// TIA Portal V20 export
// export: Created 2025-12-01T14:57:25.6351868Z, ExportSetting None, DisplayName Totally Integrated Automation Portal, DisplayVersion V20 Update 3, DisplayName TIA Portal Openness, DisplayVersion V20 Update 3, DisplayName TIA Portal Version Control Interface, DisplayVersion V20 Update 3, DisplayName STEP 7 Professional, DisplayVersion V20 Update 3, DisplayName STEP 7 Safety, DisplayVersion V20 Update 2, DisplayName WinCC Basic/Comfort/Advanced, DisplayVersion V20 Update 3, DisplayName WinCC Professional, DisplayVersion V20 Update 3, DisplayName WinCC Unified, DisplayVersion V20 Update 3
FUNCTION_BLOCK "FB483_Interlock_IKPAL_Paletas"   // FB483, LAD
{ S7_Optimized_Access := 'FALSE' }
// stored: AutoNumber false, SetENOAutomatically false
   VAR_INPUT
      MesaPreformado : UInt;
      MesaVacios : UInt;
      MesaPaleta : UInt;
      Dir_Inicial : UInt;
      Nodo_OK : Bool;
      AvisoPreformado_PRV : Bool;
      OrdenMarchaPreformado_PRV : Bool;
      AvisoPreformado_PRV_Manual_AV : Bool;
      AvisoPreformado_PRV_Manual_Ret : Bool;
      PermisoExtenderHorquilla : Bool;
      PermisoCentrarHorquilla : Bool;
      MaquetaArriba : Bool;
      MaquetaAbajo : Bool;
      PermisoPaleta_NXT : Bool;
      FinPaleta_NXT : Bool;
      PermisoPaleta_NXT_Manual_Av : Bool;
      PermisoPaleta_NXT_Manual_Ret : Bool;
      PermisoÂperturaPuertas : Bool;
   END_VAR
   VAR_OUTPUT
      EstadoIKPAL : "EstadoZona";
      PermisoPreformado_PRV : Bool;
      FinPreformado_PRV : Bool;
      PermisoPreformado_PRV_Manual_AV : Bool;
      PermisoPreformado_PRV_Manual_Ret : Bool;
      PeticionPaletaVacia : Bool;
      HorquillasExtendidas : Bool;
      HorquillasCentradas : Bool;
      SubirMaqueta_Manual : Bool;
      BajarMaqueta_Manual : Bool;
      AvisoPaleta_NXT : Bool;
      OrdenMarchaPaleta_NXT : Bool;
      AvisoPaleta_NXT_Manual_AV : Bool;
      AvisoPaleta_NXT_Manual_Ret : Bool;
      PeticionAperturaPuertas : Bool;
      PuertasAccesoAbiertas : Bool;
   END_VAR
   VAR
      IKPAL_PLC { S7_SetPoint := 'True'} : "Interlock_Paletas_IKPAL_PLC";
      PLC_IKPAL { S7_SetPoint := 'True'} : "Interlock_Paletas_PLC_IKPAL";
      TIM_KeepAlive { S7_SetPoint := 'True'} : TON_TIME;
      Var_MesaPreformado : Struct
         ControlUT { S7_SetPoint := 'True'} : "UDT_UTs_Control";
         DatosUT { S7_SetPoint := 'True'} : "UDT_UTs_Datos";
         EtiquetaUT { S7_SetPoint := 'True'} : "UDT_UTs_Etiqueta";
      END_STRUCT;
      Var_MesaVacios : Struct
         ControlUT { S7_SetPoint := 'True'} : "UDT_UTs_Control";
         DatosUT { S7_SetPoint := 'True'} : "UDT_UTs_Datos";
         EtiquetaUT { S7_SetPoint := 'True'} : "UDT_UTs_Etiqueta";
      END_STRUCT;
      UT_MesaPreformado { ExternalAccessible := 'False'; ExternalVisible := 'False'; ExternalWritable := 'False'} : UInt;
      CotaAlturaPreformado : UInt;
      Matricula_Preformado : Array[1..10] of Byte;
      Mckey_Preformado : Array[1..8] of Byte;
      UT_MesaVacios { ExternalAccessible := 'False'; ExternalVisible := 'False'; ExternalWritable := 'False'} : UInt;
      Matricula_Vacios : Array[1..10] of Byte;
      Mckey_Vacios : Array[1..8] of Byte;
      Matricula_Paleta : Array[1..10] of Byte;
      Mckey_Paleta : Array[1..8] of Byte;
      NumMckey_Paleta : DInt;
      IdentificadorUT_Paleta : UDInt;
      MemoKeepAlive : Bool;
      ExisteUT_Preformado : Bool;
      ExisteUT_Vacios : Bool;
   END_VAR
   VAR_TEMP
      EstadoMesaPreformado : "EstadoZona";
      EstadoMesaVacios : "EstadoZona";
      EstadoMesaPaleta : "EstadoZona";
      EstadoVIMesaPreformado : "EstadosMesa";
      EstadoVIMesaVacios : "EstadosMesa";
      EstadoVIMesaPaleta : "EstadosMesa";
      Interlock_Entradas : "Interlock_Paletas_IKPAL_PLC";
      Interlock_Salidas : "Interlock_Paletas_PLC_IKPAL";
      Guardar_AR1 : DWord;
      Guardar_AR2 : DWord;
      P_Entradas : Any;
      P_Salidas : Any;
      P_L_Entradas : Any;
      P_L_Salidas : Any;
      P_DI_Entradas : Any;
      P_DI_Salidas : Any;
      P_AnyTemporal : Any;
      P_Temporal : DWord;
      DBInstancia : Word;
      NumeroUT : UInt;
      LongMatricula : UInt;
      LongMckey : UInt;
      LongEntradas : UInt;
      LongSalidas : UInt;
      DBOrigen : UInt;
      DBDestino : UInt;
      OffsetOrigen : UInt;
      OffsetDestino : UInt;
      P_Origen : DWord;
      P_Destino : DWord;
      Valor : UDInt;
      Indice : UInt;
      IndiceMatricula : UInt;
      ReturnValor : Int;
      Cero : Byte;
      ErrorMaquinaAsociada : Bool;
      FlancoKeepAlive : Bool;
   END_VAR
   VAR_TEMP   // added for the SCL form of the ladder/FBD networks
      _w1 : Bool;
      _w2 : Bool;
   END_VAR
BEGIN

REGION Network 1: INICIALIZAR
END_REGION

REGION Network 2: INICIALIZAR - Recoger las Variables de Estado de la Mesa de Preformado
   // Se recoge - Estado_CBx
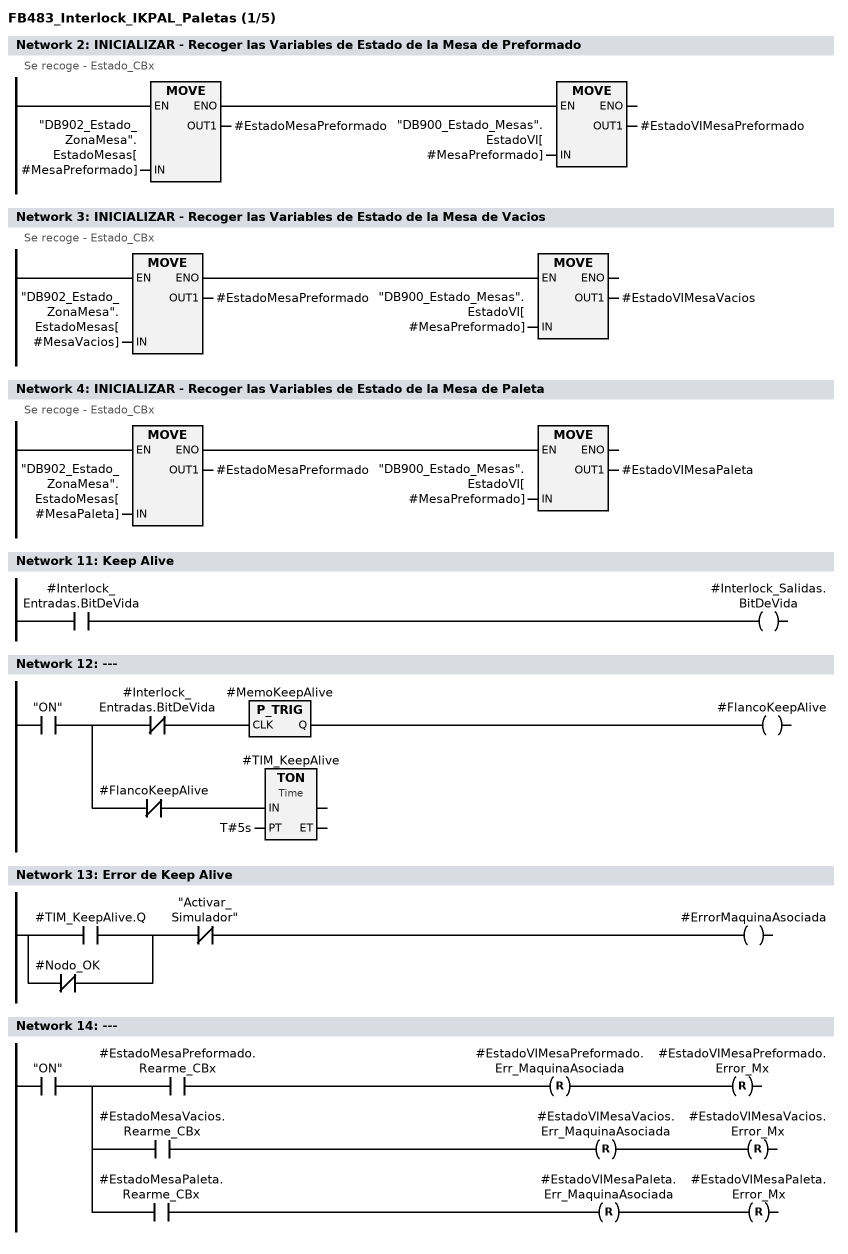
   RUNG wire#powerrail
      Move(in := "DB902_Estado_ZonaMesa".EstadoMesas[#MesaPreformado], out1 => #EstadoMesaPreformado)
      Move(in := "DB900_Estado_Mesas".EstadoVI[#MesaPreformado], out1 => #EstadoVIMesaPreformado)
   END_RUNG
   // the same network as SCL:
   #EstadoMesaPreformado := "DB902_Estado_ZonaMesa".EstadoMesas[#MesaPreformado];
   #EstadoVIMesaPreformado := "DB900_Estado_Mesas".EstadoVI[#MesaPreformado];
END_REGION

REGION Network 3: INICIALIZAR - Recoger las Variables de Estado de la Mesa de Vacios
   // Se recoge - Estado_CBx
   RUNG wire#powerrail
      Move(in := "DB902_Estado_ZonaMesa".EstadoMesas[#MesaVacios], out1 => #EstadoMesaPreformado)
      Move(in := "DB900_Estado_Mesas".EstadoVI[#MesaPreformado], out1 => #EstadoVIMesaVacios)
   END_RUNG
   // the same network as SCL:
   #EstadoMesaPreformado := "DB902_Estado_ZonaMesa".EstadoMesas[#MesaVacios];
   #EstadoVIMesaVacios := "DB900_Estado_Mesas".EstadoVI[#MesaPreformado];
END_REGION

REGION Network 4: INICIALIZAR - Recoger las Variables de Estado de la Mesa de Paleta
   // Se recoge - Estado_CBx
   RUNG wire#powerrail
      Move(in := "DB902_Estado_ZonaMesa".EstadoMesas[#MesaPaleta], out1 => #EstadoMesaPreformado)
      Move(in := "DB900_Estado_Mesas".EstadoVI[#MesaPreformado], out1 => #EstadoVIMesaPaleta)
   END_RUNG
   // the same network as SCL:
   #EstadoMesaPreformado := "DB902_Estado_ZonaMesa".EstadoMesas[#MesaPaleta];
   #EstadoVIMesaPaleta := "DB900_Estado_Mesas".EstadoVI[#MesaPreformado];
END_REGION

NETWORK
TITLE = Inicializar Variables Internas del Programa
//////////////////////////////////////////////////////////////////////////////
/// Inicializar las variables que necesita la FB

      L     56;  // Longitud de las Entradas
      T     #LongEntradas;
      L     56;  // Longitud de las Salidas
      T     #LongSalidas;
      L     10;  // Longitud de la Matricula
      T     #LongMatricula;
      L     8;  // Longitud del Mckey
      T     #LongMckey;

      L     DINO;  // Numero del DB de Instancia
      T     #DBInstancia;




NETWORK
TITLE = Preparacion de Punteros Any de las Entradas y Salidas
//////////////////////////////////////////////////////////////////////////////

      TAR1  #Guardar_AR1;  // Guardar AR1


//////////////////////////////////////////////////////////////////////////////
/// Puntero Any a las Entradas y Salidas (Temporales)

      LAR1  P##P_L_Entradas;  // - Any - Entradas del interlock
      L     B#16#10;  //   10H para S7
      T     LB [AR1, P#0.0];
      L     B#16#2;  //   Tipo de Datos (BYTE)
      T     LB [AR1, P#1.0];
      L     #LongEntradas;  //   Cantidad de datos
      T     LW [AR1, P#2.0];
      L     0;  //   Numero de DB (Temporal = 0)
      T     LW [AR1, P#4.0];
      L     P##Interlock_Entradas;  //   Direccion de Inicio
      T     LD [AR1, P#6.0];
      L     B#16#87;  //   El Area de Memoria = Temporal (Nota: No 86)
      T     LB [AR1, P#6.0];


      LAR1  P##P_L_Salidas;  // - Any - Salidas del interlock
      L     B#16#10;  //   10H para S7
      T     LB [AR1, P#0.0];
      L     B#16#2;  //   Tipo de Datos (BYTE)
      T     LB [AR1, P#1.0];
      L     #LongSalidas;  //   Cantidad de datos
      T     LW [AR1, P#2.0];
      L     0;  //   Numero de DB (Temporal = 0)
      T     LW [AR1, P#4.0];
      L     P##Interlock_Salidas;  //   Direccion de Inicio
      T     LD [AR1, P#6.0];
      L     B#16#87;  //   El Area de Memoria = Temporal (Nota: No 86)
      T     LB [AR1, P#6.0];


//////////////////////////////////////////////////////////////////////////////
/// Puntero Any a las Entradas y Salidas (DB de Instancia)

      LAR1  P##P_DI_Entradas;  // - Any - Entradas del interlock
      L     B#16#10;  //   10H para S7
      T     LB [AR1, P#0.0];
      L     B#16#2;  //   Tipo de Datos (BYTE)
      T     LB [AR1, P#1.0];
      L     #LongEntradas;  //   Cantidad de datos
      T     LW [AR1, P#2.0];
      L     #DBInstancia;  //   Numero de DB de Instancia
      T     LW [AR1, P#4.0];
      L     P##IKPAL_PLC;  //   Direccion de Inicio
      T     LD [AR1, P#6.0];
      L     B#16#84;  //   El Area de Memoria = DB Instancia
      T     LB [AR1, P#6.0];

      LAR1  P##P_DI_Salidas;  // - Any - Salidas del interlock
      L     B#16#10;  //   10H para S7
      T     LB [AR1, P#0.0];
      L     B#16#2;  //   Tipo de Datos (BYTE)
      T     LB [AR1, P#1.0];
      L     #LongSalidas;  //   Cantidad de datos
      T     LW [AR1, P#2.0];
      L     #DBInstancia;  //   Numero de DB de Instancia
      T     LW [AR1, P#4.0];
      L     P##PLC_IKPAL;  //   Direccion de Inicio
      T     LD [AR1, P#6.0];
      L     B#16#84;  //   El Area de Memoria = DB Instancia
      T     LB [AR1, P#6.0];


//////////////////////////////////////////////////////////////////////////////
/// Puntero Any - De Lectura y Escritura de QUBIQA

      LAR1  P##P_Entradas;  // - Any - Entradas del interlock
      L     B#16#10;  //   10H para S7
      T     LB [AR1, P#0.0];
      L     B#16#2;  //   Tipo de Datos (BYTE)
      T     LB [AR1, P#1.0];
      L     #LongEntradas;  //   Cantidad de datos
      T     LW [AR1, P#2.0];
      L     0;  //   Numero de DB (Temporal = 0)
      T     LW [AR1, P#4.0];
      L     #Dir_Inicial;  //   Direccion de Inicio
      SLD   3;
      T     LD [AR1, P#6.0];
      L     B#16#81;  //   El Area de Memoria = Entradas
      T     LB [AR1, P#6.0];

      LAR1  P##P_Salidas;  // - Any - Entradas del interlock
      L     B#16#10;  //   10H para S7
      T     LB [AR1, P#0.0];
      L     B#16#2;  //   Tipo de Datos (BYTE)
      T     LB [AR1, P#1.0];
      L     #LongSalidas;  //   Cantidad de datos
      T     LW [AR1, P#2.0];
      L     0;  //   Numero de DB (Temporal = 0)
      T     LW [AR1, P#4.0];
      L     #Dir_Inicial;  //   Direccion de Inicio
      SLD   3;
      T     LD [AR1, P#6.0];
      L     B#16#82;  //   El Area de Memoria = Salidas
      T     LB [AR1, P#6.0];

//////////////////////////////////////////////////////////////////////////////

      LAR1  #Guardar_AR1;  // Recuperar AR1



NETWORK
TITLE = Inicializacion de las Entradas y Salidas
//////////////////////////////////////////////////////////////////////////////
/// Inicializar el interlock (Variables Temporales)

      L     0;
      T     #Cero;

      CALL  FILL
      ( BVAL    := #Cero,
        RET_VAL := #ReturnValor,
        BLK     := #P_L_Entradas
      );  // Inicializo las Entradas

      CALL  FILL
      ( BVAL    := #Cero,
        RET_VAL := #ReturnValor,
        BLK     := #P_L_Salidas
      );  // Inicializo las Salidas



NETWORK
TITLE = Lectura de las Entradas
//////////////////////////////////////////////////////////////////////////////
/// Lectura de las Entradas

      SET;  // Comprobacion del Nodo
      AN    #Nodo_OK;
      AN    "Activar_Simulador";
      JC    NoLeerInterlock;

      CALL  UBLKMOV
      ( SRCBLK  := #P_Entradas,
        RET_VAL := #ReturnValor,
        DSTBLK  := #P_L_Entradas
      );


//////////////////////////////////////////////////////////////////////////////
/// Final Lectura de las Entradas

NoLeerInterlock:NOP   0;

      CALL  UBLKMOV
      ( SRCBLK  := #P_L_Entradas,
        RET_VAL := #ReturnValor,
        DSTBLK  := #P_DI_Entradas
      );  // Guardar el DB de Instancia



NETWORK
TITLE = Leer Datos de la UT de la Mesa de Preformado
//////////////////////////////////////////////////////////////////////////////
/// Incializacion inicial
      SET;  // De Inicio no existe UT
      R     #ExisteUT_Preformado;

      L     0;
      T     #UT_MesaPreformado;

      L     0;
      T     #Cero;
      CALL  FILL
      ( BVAL    := #Cero,
        RET_VAL := #ReturnValor,
        BLK     := #Var_MesaPreformado
      );

      SET;
      L     #MesaPreformado;  // Existe Mesa de Preformado ?
      L     0;
      ==I;
      JC    NoExiteUT_Preformado;


//////////////////////////////////////////////////////////////////////////////
/// Se mira si existe UT
      L     "DB810_ColasMesas".Colas[#MesaPreformado].UT_PrimeraMesa;
      T     #NumeroUT;
      L     0;
      ==I;
      JC    NoExiteUT_Preformado;

      SET;  // Existe UT en la Mesa
      S     #ExisteUT_Preformado;

      L     #NumeroUT;
      T     #UT_MesaPreformado;

      CALL  BLKMOV
      ( SRCBLK  := "DB812_UTs_Control".UT[#UT_MesaPreformado],
        RET_VAL := #ReturnValor,
        DSTBLK  := #Var_MesaPreformado.ControlUT
      );
      CALL  BLKMOV
      ( SRCBLK  := "DB815_UTs_Datos".UT[#UT_MesaPreformado],
        RET_VAL := #ReturnValor,
        DSTBLK  := #Var_MesaPreformado.DatosUT
      );
      CALL  BLKMOV
      ( SRCBLK  := "DB814_UTs_Etiqueta".UT[#MesaPreformado],
        RET_VAL := #ReturnValor,
        DSTBLK  := #Var_MesaPreformado.EtiquetaUT
      );


//////////////////////////////////////////////////////////////////////////////
/// Inicializo los datos de la UT que necesita el Interlock de IKPAL
      CALL  FILL
      ( BVAL    := #Cero,
        RET_VAL := #ReturnValor,
        BLK     := #Mckey_Preformado
      );  // Inicializo el Mckey

      CALL  FILL
      ( BVAL    := #Cero,
        RET_VAL := #ReturnValor,
        BLK     := #Matricula_Preformado
      );  // Inicializo la Matricula

//////////////////////////////////////////////////////////////////////////////
/// Copia el Cota Altura de la UT para el Interlock con IKPAL
      L     "DB815_UTs_Datos".UT[#UT_MesaPreformado].CotaAltura;
      T     #CotaAlturaPreformado;

//////////////////////////////////////////////////////////////////////////////
/// Copia el Mckey de la UT para el Interlock con IKPAL
      L     "DB812_UTs_Control".UT[#UT_MesaPreformado].Mckey;
      T     #Valor;

      L     #DBInstancia;
      T     #DBDestino;
      L     P##Mckey_Preformado;
      T     #P_Destino;
      SRD   3;
      L     #LongMckey;
      +I;
      L     1;
      -I;
      T     #OffsetDestino;

      CALL  "FC891_EtiqDInt_EtiqChar"
      ( DB_String   := #DBDestino,
        Long_String := #LongMckey,
        Offset_Ini  := #OffsetDestino,
        Valor       := #Valor
      );

      L     #LongMckey;
Copia_MckeyPreformado:T     #Indice;

      OPN   DB [#DBDestino];
      L     DBB [#P_Destino];
      L     '0';
      -I;
      OPN   DB [#DBDestino];
      T     DBB [#P_Destino];

      L     #P_Destino;
      L     P#1.0;
      +D;
      T     #P_Destino;

      L     #Indice;
      LOOP  Copia_MckeyPreformado;


//////////////////////////////////////////////////////////////////////////////
/// Copia la Matricula de la UT para el Interlock con IKPAL
      L     0;
      T     #IndiceMatricula;

      L     #DBInstancia;
      T     #DBDestino;
      L     P##Matricula_Preformado;
      T     #P_Destino;

      L     #LongMatricula;
Copia_MatriculaPreformado:T     #Indice;

      L     "DB814_UTs_Etiqueta".UT[#UT_MesaPreformado].Etiqueta[#IndiceMatricula];
      L     '0';
      -I;
      OPN   DB [#DBDestino];
      T     DBB [#P_Destino];

      L     #IndiceMatricula;
      L     1;
      +I;
      T     #IndiceMatricula;

      L     #P_Destino;
      L     P#1.0;
      +D;
      T     #P_Destino;

      L     #Indice;
      LOOP  Copia_MatriculaPreformado;


//////////////////////////////////////////////////////////////////////////////
NoExiteUT_Preformado:NOP   0;  // Final de la Lectura de Datos



NETWORK
TITLE = Leer Datos de la UT de la Mesa de Vacios
//////////////////////////////////////////////////////////////////////////////
/// Incializacion inicial
      SET;  // De Inicio no existe UT
      R     #ExisteUT_Vacios;

      L     0;
      T     #Cero;
      CALL  FILL
      ( BVAL    := #Cero,
        RET_VAL := #ReturnValor,
        BLK     := #Var_MesaVacios
      );


      SET;
      L     #MesaVacios;  // Existe Mesa de Preformado ?
      L     0;
      ==I;
      JC    NoExiteUT_Vacios;


//////////////////////////////////////////////////////////////////////////////
/// Se mira si existe UT
      L     "DB810_ColasMesas".Colas[#MesaVacios].UT_PrimeraMesa;
      T     #NumeroUT;
      L     0;
      ==I;
      JC    NoExiteUT_Vacios;

      SET;  // Existe UT en la Mesa
      S     #ExisteUT_Vacios;

      L     #NumeroUT;
      T     #UT_MesaVacios;

      CALL  BLKMOV
      ( SRCBLK  := "DB812_UTs_Control".UT[#UT_MesaVacios],
        RET_VAL := #ReturnValor,
        DSTBLK  := #Var_MesaVacios.ControlUT
      );
      CALL  BLKMOV
      ( SRCBLK  := "DB815_UTs_Datos".UT[#UT_MesaVacios],
        RET_VAL := #ReturnValor,
        DSTBLK  := #Var_MesaVacios.DatosUT
      );
      CALL  BLKMOV
      ( SRCBLK  := "DB814_UTs_Etiqueta".UT[#MesaVacios],
        RET_VAL := #ReturnValor,
        DSTBLK  := #Var_MesaVacios.EtiquetaUT
      );


//////////////////////////////////////////////////////////////////////////////
/// Inicializo los datos de la UT que necesita el Interlock de IKPAL
      CALL  FILL
      ( BVAL    := #Cero,
        RET_VAL := #ReturnValor,
        BLK     := #Mckey_Vacios
      );  // Inicializo el Mckey

      CALL  FILL
      ( BVAL    := #Cero,
        RET_VAL := #ReturnValor,
        BLK     := #Matricula_Vacios
      );  // Inicializo la Matricula


//////////////////////////////////////////////////////////////////////////////
/// Copia el Mckey de la UT para el Interlock con IKPAL
      L     "DB812_UTs_Control".UT[#UT_MesaVacios].Mckey;
      T     #Valor;

      L     #DBInstancia;
      T     #DBDestino;
      L     P##Mckey_Vacios;
      T     #P_Destino;
      SRD   3;
      L     #LongMckey;
      +I;
      L     1;
      -I;
      T     #OffsetDestino;

      CALL  "FC891_EtiqDInt_EtiqChar"
      ( DB_String   := #DBDestino,
        Long_String := #LongMckey,
        Offset_Ini  := #OffsetDestino,
        Valor       := #Valor
      );

      L     #LongMckey;
Copia_MckeyVacios:T     #Indice;

      OPN   DB [#DBDestino];
      L     DBB [#P_Destino];
      L     '0';
      -I;
      OPN   DB [#DBDestino];
      T     DBB [#P_Destino];

      L     #P_Destino;
      L     P#1.0;
      +D;
      T     #P_Destino;

      L     #Indice;
      LOOP  Copia_MckeyVacios;


//////////////////////////////////////////////////////////////////////////////
/// Copia la Matricula de la UT para el Interlock con IKPA
      L     0;
      T     #IndiceMatricula;

      L     #DBInstancia;
      T     #DBDestino;
      L     P##Matricula_Vacios;
      T     #P_Destino;

      L     #LongMatricula;
Copia_MatriculaVacios:T     #Indice;

      L     "DB814_UTs_Etiqueta".UT[#UT_MesaVacios].Etiqueta[#IndiceMatricula];
      L     '0';
      -I;
      OPN   DB [#DBDestino];
      T     DBB [#P_Destino];

      L     #IndiceMatricula;
      L     1;
      +I;
      T     #IndiceMatricula;

      L     #P_Destino;
      L     P#1.0;
      +D;
      T     #P_Destino;

      L     #Indice;
      LOOP  Copia_MatriculaVacios;


//////////////////////////////////////////////////////////////////////////////
NoExiteUT_Vacios:NOP   0;  // Final de la Lectura de Datos



REGION Network 11: Keep Alive
   RUNG wire#powerrail
      Contact( #Interlock_Entradas.BitDeVida )
      Coil( #Interlock_Salidas.BitDeVida )
   END_RUNG
   // the same network as SCL:
   #Interlock_Salidas.BitDeVida := #Interlock_Entradas.BitDeVida;
END_REGION

REGION Network 12: ---
   RUNG wire#powerrail
      Contact( "ON" )
      wire#w1
      I_Contact( #Interlock_Entradas.BitDeVida )
      P_Trig( #MemoKeepAlive )
      Coil( #FlancoKeepAlive )
   END_RUNG
   RUNG wire#w1
      I_Contact( #FlancoKeepAlive )
      { S7_Templates := "time_type := Time" } #TIM_KeepAlive.TON(pt := T#5s, et =>)
   END_RUNG
   // the same network as SCL:
   #_w1 := "ON" AND NOT #Interlock_Entradas.BitDeVida;
   #_w2 := #_w1 AND NOT #MemoKeepAlive;   // rising edge
   #MemoKeepAlive := #_w1;
   #FlancoKeepAlive := #_w2;
   #TIM_KeepAlive(IN := "ON" AND NOT #FlancoKeepAlive, PT := T#5s);   // TON
END_REGION

REGION Network 13: Error de Keep Alive
   RUNG wire#powerrail
      Contact( #TIM_KeepAlive.Q )
      wire#w1
      I_Contact( "Activar_Simulador" )
      Coil( #ErrorMaquinaAsociada )
   END_RUNG
   RUNG wire#powerrail
      I_Contact( #Nodo_OK )
   END_RUNG wire#w1
   // the same network as SCL:
   #ErrorMaquinaAsociada := (#TIM_KeepAlive.Q OR NOT #Nodo_OK) AND NOT "Activar_Simulador";
END_REGION

REGION Network 14: ---
   RUNG wire#powerrail
      Contact( "ON" )
      wire#w1
      Contact( #EstadoMesaPreformado.Rearme_CBx )
      R_Coil( #EstadoVIMesaPreformado.Err_MaquinaAsociada )
      R_Coil( #EstadoVIMesaPreformado.Error_Mx )
   END_RUNG
   RUNG wire#w1
      Contact( #EstadoMesaVacios.Rearme_CBx )
      R_Coil( #EstadoVIMesaVacios.Err_MaquinaAsociada )
      R_Coil( #EstadoVIMesaVacios.Error_Mx )
   END_RUNG
   RUNG wire#w1
      Contact( #EstadoMesaPaleta.Rearme_CBx )
      R_Coil( #EstadoVIMesaPaleta.Err_MaquinaAsociada )
      R_Coil( #EstadoVIMesaPaleta.Error_Mx )
   END_RUNG
   // the same network as SCL:
   IF "ON" AND #EstadoMesaPreformado.Rearme_CBx THEN
       #EstadoVIMesaPreformado.Err_MaquinaAsociada := FALSE;
       #EstadoVIMesaPreformado.Error_Mx := FALSE;
   END_IF;
   IF "ON" AND #EstadoMesaVacios.Rearme_CBx THEN
       #EstadoVIMesaVacios.Err_MaquinaAsociada := FALSE;
       #EstadoVIMesaVacios.Error_Mx := FALSE;
   END_IF;
   IF "ON" AND #EstadoMesaPaleta.Rearme_CBx THEN
       #EstadoVIMesaPaleta.Err_MaquinaAsociada := FALSE;
       #EstadoVIMesaPaleta.Error_Mx := FALSE;
   END_IF;
END_REGION

REGION Network 15: ---
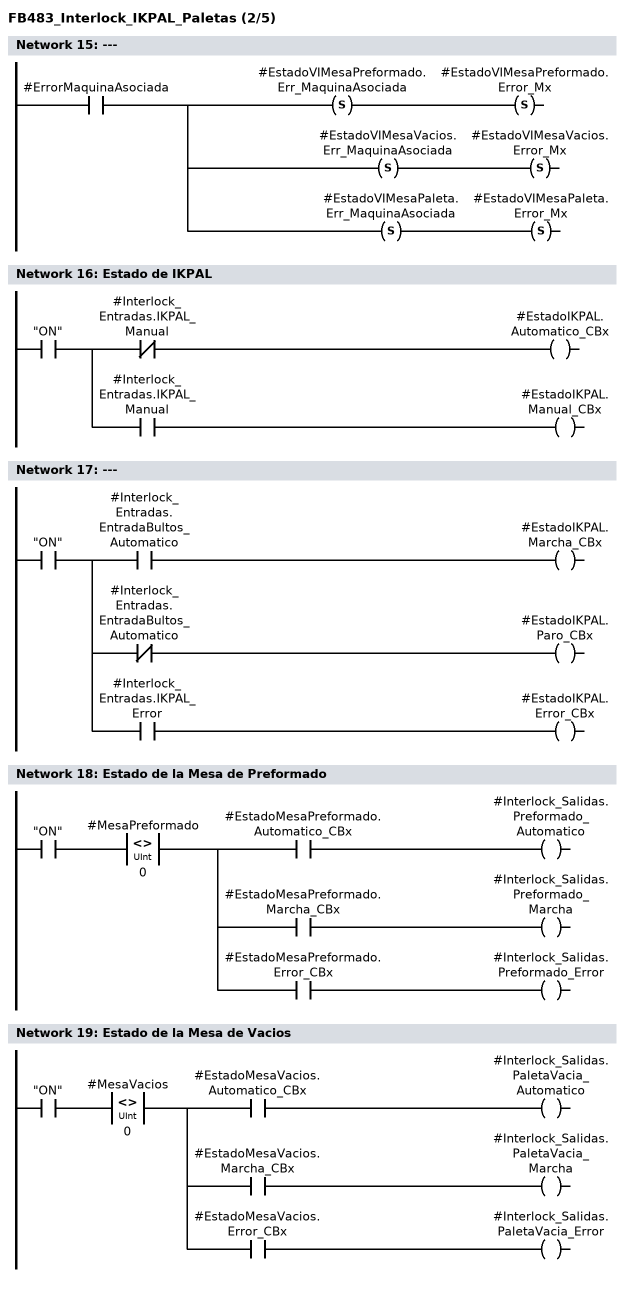
   RUNG wire#powerrail
      Contact( #ErrorMaquinaAsociada )
      wire#w1
      S_Coil( #EstadoVIMesaPreformado.Err_MaquinaAsociada )
      S_Coil( #EstadoVIMesaPreformado.Error_Mx )
   END_RUNG
   RUNG wire#w1
      S_Coil( #EstadoVIMesaVacios.Err_MaquinaAsociada )
      S_Coil( #EstadoVIMesaVacios.Error_Mx )
   END_RUNG
   RUNG wire#w1
      S_Coil( #EstadoVIMesaPaleta.Err_MaquinaAsociada )
      S_Coil( #EstadoVIMesaPaleta.Error_Mx )
   END_RUNG
   // the same network as SCL:
   IF #ErrorMaquinaAsociada THEN
       #EstadoVIMesaPreformado.Err_MaquinaAsociada := TRUE;
       #EstadoVIMesaPreformado.Error_Mx := TRUE;
       #EstadoVIMesaVacios.Err_MaquinaAsociada := TRUE;
       #EstadoVIMesaVacios.Error_Mx := TRUE;
       #EstadoVIMesaPaleta.Err_MaquinaAsociada := TRUE;
       #EstadoVIMesaPaleta.Error_Mx := TRUE;
   END_IF;
END_REGION

REGION Network 16: Estado de IKPAL
   RUNG wire#powerrail
      Contact( "ON" )
      wire#w1
      I_Contact( #Interlock_Entradas.IKPAL_Manual )
      Coil( #EstadoIKPAL.Automatico_CBx )
   END_RUNG
   RUNG wire#w1
      Contact( #Interlock_Entradas.IKPAL_Manual )
      Coil( #EstadoIKPAL.Manual_CBx )
   END_RUNG
   // the same network as SCL:
   #EstadoIKPAL.Automatico_CBx := "ON" AND NOT #Interlock_Entradas.IKPAL_Manual;
   #EstadoIKPAL.Manual_CBx := "ON" AND #Interlock_Entradas.IKPAL_Manual;
END_REGION

REGION Network 17: ---
   RUNG wire#powerrail
      Contact( "ON" )
      wire#w1
      Contact( #Interlock_Entradas.EntradaBultos_Automatico )
      Coil( #EstadoIKPAL.Marcha_CBx )
   END_RUNG
   RUNG wire#w1
      I_Contact( #Interlock_Entradas.EntradaBultos_Automatico )
      Coil( #EstadoIKPAL.Paro_CBx )
   END_RUNG
   RUNG wire#w1
      Contact( #Interlock_Entradas.IKPAL_Error )
      Coil( #EstadoIKPAL.Error_CBx )
   END_RUNG
   // the same network as SCL:
   #EstadoIKPAL.Marcha_CBx := "ON" AND #Interlock_Entradas.EntradaBultos_Automatico;
   #EstadoIKPAL.Paro_CBx := "ON" AND NOT #Interlock_Entradas.EntradaBultos_Automatico;
   #EstadoIKPAL.Error_CBx := "ON" AND #Interlock_Entradas.IKPAL_Error;
END_REGION

REGION Network 18: Estado de la Mesa de Preformado
   RUNG wire#powerrail
      Contact( "ON" )
      { S7_Templates := "SrcType := UInt" } NE_Contact(in1 := #MesaPreformado, in2 := 0)
      wire#w1
      Contact( #EstadoMesaPreformado.Automatico_CBx )
      Coil( #Interlock_Salidas.Preformado_Automatico )
   END_RUNG
   RUNG wire#w1
      Contact( #EstadoMesaPreformado.Marcha_CBx )
      Coil( #Interlock_Salidas.Preformado_Marcha )
   END_RUNG
   RUNG wire#w1
      Contact( #EstadoMesaPreformado.Error_CBx )
      Coil( #Interlock_Salidas.Preformado_Error )
   END_RUNG
   // the same network as SCL:
   #_w1 := "ON" AND (#MesaPreformado <> 0);
   #Interlock_Salidas.Preformado_Automatico := #_w1 AND #EstadoMesaPreformado.Automatico_CBx;
   #Interlock_Salidas.Preformado_Marcha := #_w1 AND #EstadoMesaPreformado.Marcha_CBx;
   #Interlock_Salidas.Preformado_Error := #_w1 AND #EstadoMesaPreformado.Error_CBx;
END_REGION

REGION Network 19: Estado de la Mesa de Vacios
   RUNG wire#powerrail
      Contact( "ON" )
      { S7_Templates := "SrcType := UInt" } NE_Contact(in1 := #MesaVacios, in2 := 0)
      wire#w1
      Contact( #EstadoMesaVacios.Automatico_CBx )
      Coil( #Interlock_Salidas.PaletaVacia_Automatico )
   END_RUNG
   RUNG wire#w1
      Contact( #EstadoMesaVacios.Marcha_CBx )
      Coil( #Interlock_Salidas.PaletaVacia_Marcha )
   END_RUNG
   RUNG wire#w1
      Contact( #EstadoMesaVacios.Error_CBx )
      Coil( #Interlock_Salidas.PaletaVacia_Error )
   END_RUNG
   // the same network as SCL:
   #_w1 := "ON" AND (#MesaVacios <> 0);
   #Interlock_Salidas.PaletaVacia_Automatico := #_w1 AND #EstadoMesaVacios.Automatico_CBx;
   #Interlock_Salidas.PaletaVacia_Marcha := #_w1 AND #EstadoMesaVacios.Marcha_CBx;
   #Interlock_Salidas.PaletaVacia_Error := #_w1 AND #EstadoMesaVacios.Error_CBx;
END_REGION

REGION Network 20: Estado de la Mesa de la Paleta
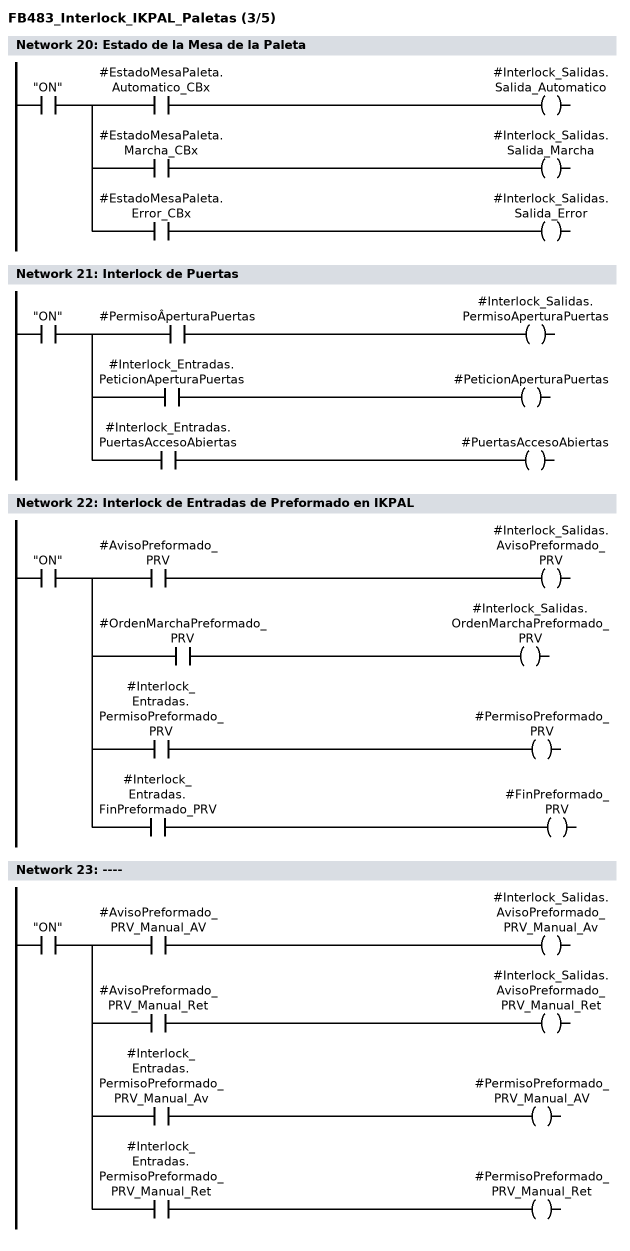
   RUNG wire#powerrail
      Contact( "ON" )
      wire#w1
      Contact( #EstadoMesaPaleta.Automatico_CBx )
      Coil( #Interlock_Salidas.Salida_Automatico )
   END_RUNG
   RUNG wire#w1
      Contact( #EstadoMesaPaleta.Marcha_CBx )
      Coil( #Interlock_Salidas.Salida_Marcha )
   END_RUNG
   RUNG wire#w1
      Contact( #EstadoMesaPaleta.Error_CBx )
      Coil( #Interlock_Salidas.Salida_Error )
   END_RUNG
   // the same network as SCL:
   #Interlock_Salidas.Salida_Automatico := "ON" AND #EstadoMesaPaleta.Automatico_CBx;
   #Interlock_Salidas.Salida_Marcha := "ON" AND #EstadoMesaPaleta.Marcha_CBx;
   #Interlock_Salidas.Salida_Error := "ON" AND #EstadoMesaPaleta.Error_CBx;
END_REGION

REGION Network 21: Interlock de Puertas
   RUNG wire#powerrail
      Contact( "ON" )
      wire#w1
      Contact( #PermisoÂperturaPuertas )
      Coil( #Interlock_Salidas.PermisoAperturaPuertas )
   END_RUNG
   RUNG wire#w1
      Contact( #Interlock_Entradas.PeticionAperturaPuertas )
      Coil( #PeticionAperturaPuertas )
   END_RUNG
   RUNG wire#w1
      Contact( #Interlock_Entradas.PuertasAccesoAbiertas )
      Coil( #PuertasAccesoAbiertas )
   END_RUNG
   // the same network as SCL:
   #Interlock_Salidas.PermisoAperturaPuertas := "ON" AND #PermisoÂperturaPuertas;
   #PeticionAperturaPuertas := "ON" AND #Interlock_Entradas.PeticionAperturaPuertas;
   #PuertasAccesoAbiertas := "ON" AND #Interlock_Entradas.PuertasAccesoAbiertas;
END_REGION

REGION Network 22: Interlock de Entradas de Preformado en IKPAL
   RUNG wire#powerrail
      Contact( "ON" )
      wire#w1
      Contact( #AvisoPreformado_PRV )
      Coil( #Interlock_Salidas.AvisoPreformado_PRV )
   END_RUNG
   RUNG wire#w1
      Contact( #OrdenMarchaPreformado_PRV )
      Coil( #Interlock_Salidas.OrdenMarchaPreformado_PRV )
   END_RUNG
   RUNG wire#w1
      Contact( #Interlock_Entradas.PermisoPreformado_PRV )
      Coil( #PermisoPreformado_PRV )
   END_RUNG
   RUNG wire#w1
      Contact( #Interlock_Entradas.FinPreformado_PRV )
      Coil( #FinPreformado_PRV )
   END_RUNG
   // the same network as SCL:
   #Interlock_Salidas.AvisoPreformado_PRV := "ON" AND #AvisoPreformado_PRV;
   #Interlock_Salidas.OrdenMarchaPreformado_PRV := "ON" AND #OrdenMarchaPreformado_PRV;
   #PermisoPreformado_PRV := "ON" AND #Interlock_Entradas.PermisoPreformado_PRV;
   #FinPreformado_PRV := "ON" AND #Interlock_Entradas.FinPreformado_PRV;
END_REGION

REGION Network 23: ----
   RUNG wire#powerrail
      Contact( "ON" )
      wire#w1
      Contact( #AvisoPreformado_PRV_Manual_AV )
      Coil( #Interlock_Salidas.AvisoPreformado_PRV_Manual_Av )
   END_RUNG
   RUNG wire#w1
      Contact( #AvisoPreformado_PRV_Manual_Ret )
      Coil( #Interlock_Salidas.AvisoPreformado_PRV_Manual_Ret )
   END_RUNG
   RUNG wire#w1
      Contact( #Interlock_Entradas.PermisoPreformado_PRV_Manual_Av )
      Coil( #PermisoPreformado_PRV_Manual_AV )
   END_RUNG
   RUNG wire#w1
      Contact( #Interlock_Entradas.PermisoPreformado_PRV_Manual_Ret )
      Coil( #PermisoPreformado_PRV_Manual_Ret )
   END_RUNG
   // the same network as SCL:
   #Interlock_Salidas.AvisoPreformado_PRV_Manual_Av := "ON" AND #AvisoPreformado_PRV_Manual_AV;
   #Interlock_Salidas.AvisoPreformado_PRV_Manual_Ret := "ON" AND #AvisoPreformado_PRV_Manual_Ret;
   #PermisoPreformado_PRV_Manual_AV := "ON" AND #Interlock_Entradas.PermisoPreformado_PRV_Manual_Av;
   #PermisoPreformado_PRV_Manual_Ret := "ON" AND #Interlock_Entradas.PermisoPreformado_PRV_Manual_Ret;
END_REGION

NETWORK
TITLE = ----
//////////////////////////////////////////////////////////////////
/// Copia de los datos de la Mesa de Preformado para IKPAL

      AN    #ExisteUT_Preformado;
      JC    FinalCopiaDatos_Preformado_IKPAL;

      L     #CotaAlturaPreformado;
      T     #Interlock_Salidas.CotaAlturaPreformado;

      CALL  UBLKMOV
      ( SRCBLK  := #Mckey_Preformado,
        RET_VAL := #ReturnValor,
        DSTBLK  := #Interlock_Salidas.MckeyPreformado
      );
      CALL  UBLKMOV
      ( SRCBLK  := #Matricula_Preformado,
        RET_VAL := #ReturnValor,
        DSTBLK  := #Interlock_Salidas.MatriculaPreformado
      );

FinalCopiaDatos_Preformado_IKPAL:NOP   0;



REGION Network 25: Interlock de Entradas de Vacios en IKPAL
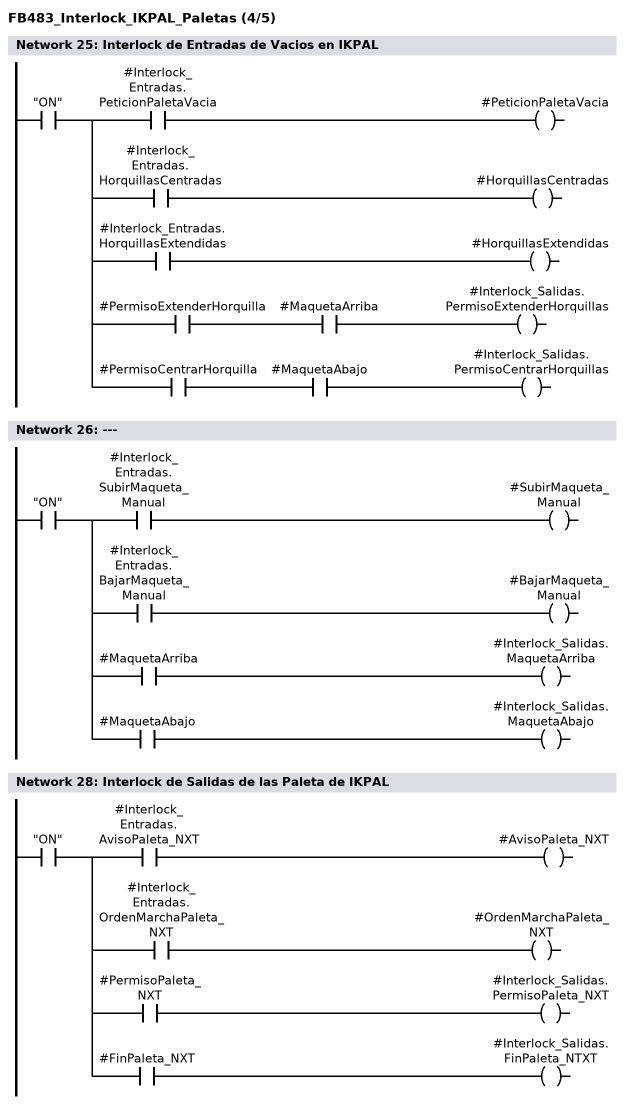
   RUNG wire#powerrail
      Contact( "ON" )
      wire#w1
      Contact( #Interlock_Entradas.PeticionPaletaVacia )
      Coil( #PeticionPaletaVacia )
   END_RUNG
   RUNG wire#w1
      Contact( #Interlock_Entradas.HorquillasCentradas )
      Coil( #HorquillasCentradas )
   END_RUNG
   RUNG wire#w1
      Contact( #Interlock_Entradas.HorquillasExtendidas )
      Coil( #HorquillasExtendidas )
   END_RUNG
   RUNG wire#w1
      Contact( #PermisoExtenderHorquilla )
      Contact( #MaquetaArriba )
      Coil( #Interlock_Salidas.PermisoExtenderHorquillas )
   END_RUNG
   RUNG wire#w1
      Contact( #PermisoCentrarHorquilla )
      Contact( #MaquetaAbajo )
      Coil( #Interlock_Salidas.PermisoCentrarHorquillas )
   END_RUNG
   // the same network as SCL:
   #PeticionPaletaVacia := "ON" AND #Interlock_Entradas.PeticionPaletaVacia;
   #HorquillasCentradas := "ON" AND #Interlock_Entradas.HorquillasCentradas;
   #HorquillasExtendidas := "ON" AND #Interlock_Entradas.HorquillasExtendidas;
   #Interlock_Salidas.PermisoExtenderHorquillas := "ON" AND #PermisoExtenderHorquilla AND #MaquetaArriba;
   #Interlock_Salidas.PermisoCentrarHorquillas := "ON" AND #PermisoCentrarHorquilla AND #MaquetaAbajo;
END_REGION

REGION Network 26: ---
   RUNG wire#powerrail
      Contact( "ON" )
      wire#w1
      Contact( #Interlock_Entradas.SubirMaqueta_Manual )
      Coil( #SubirMaqueta_Manual )
   END_RUNG
   RUNG wire#w1
      Contact( #Interlock_Entradas.BajarMaqueta_Manual )
      Coil( #BajarMaqueta_Manual )
   END_RUNG
   RUNG wire#w1
      Contact( #MaquetaArriba )
      Coil( #Interlock_Salidas.MaquetaArriba )
   END_RUNG
   RUNG wire#w1
      Contact( #MaquetaAbajo )
      Coil( #Interlock_Salidas.MaquetaAbajo )
   END_RUNG
   // the same network as SCL:
   #SubirMaqueta_Manual := "ON" AND #Interlock_Entradas.SubirMaqueta_Manual;
   #BajarMaqueta_Manual := "ON" AND #Interlock_Entradas.BajarMaqueta_Manual;
   #Interlock_Salidas.MaquetaArriba := "ON" AND #MaquetaArriba;
   #Interlock_Salidas.MaquetaAbajo := "ON" AND #MaquetaAbajo;
END_REGION

NETWORK
TITLE = ----
//////////////////////////////////////////////////////////////////
/// Copia de los datos de la Mesa de Vacios para IKPAL

      AN    #ExisteUT_Vacios;
      JC    FinalCopiaDatos_Vacios_IKPAL;

      CALL  UBLKMOV
      ( SRCBLK  := #Mckey_Vacios,
        RET_VAL := #ReturnValor,
        DSTBLK  := #Interlock_Salidas.MckeyPaletaVacia
      );
      CALL  UBLKMOV
      ( SRCBLK  := #Matricula_Vacios,
        RET_VAL := #ReturnValor,
        DSTBLK  := #Interlock_Salidas.MatriculaPaletaVacia
      );

FinalCopiaDatos_Vacios_IKPAL:NOP   0;



REGION Network 28: Interlock de Salidas de las Paleta de IKPAL
   RUNG wire#powerrail
      Contact( "ON" )
      wire#w1
      Contact( #Interlock_Entradas.AvisoPaleta_NXT )
      Coil( #AvisoPaleta_NXT )
   END_RUNG
   RUNG wire#w1
      Contact( #Interlock_Entradas.OrdenMarchaPaleta_NXT )
      Coil( #OrdenMarchaPaleta_NXT )
   END_RUNG
   RUNG wire#w1
      Contact( #PermisoPaleta_NXT )
      Coil( #Interlock_Salidas.PermisoPaleta_NXT )
   END_RUNG
   RUNG wire#w1
      Contact( #FinPaleta_NXT )
      Coil( #Interlock_Salidas.FinPaleta_NTXT )
   END_RUNG
   // the same network as SCL:
   #AvisoPaleta_NXT := "ON" AND #Interlock_Entradas.AvisoPaleta_NXT;
   #OrdenMarchaPaleta_NXT := "ON" AND #Interlock_Entradas.OrdenMarchaPaleta_NXT;
   #Interlock_Salidas.PermisoPaleta_NXT := "ON" AND #PermisoPaleta_NXT;
   #Interlock_Salidas.FinPaleta_NTXT := "ON" AND #FinPaleta_NXT;
END_REGION

REGION Network 29: ---
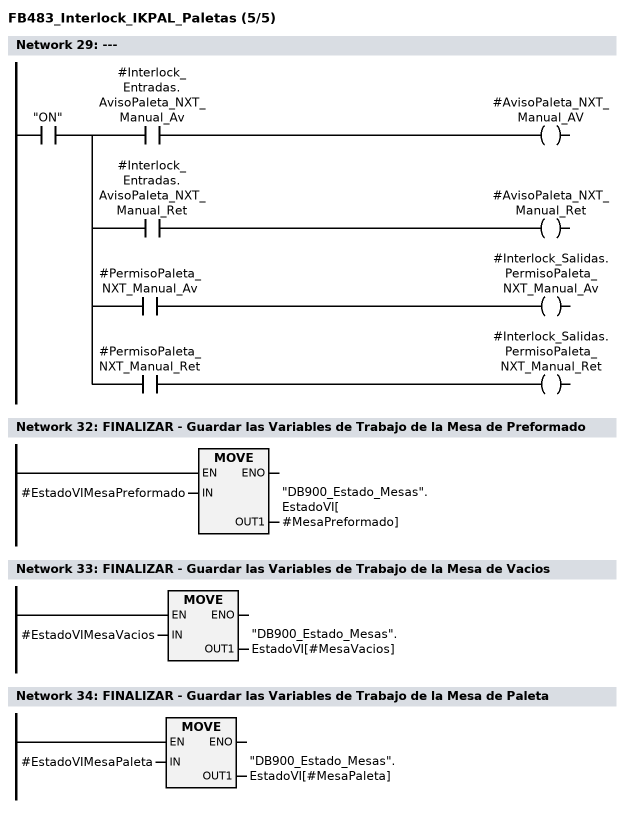
   RUNG wire#powerrail
      Contact( "ON" )
      wire#w1
      Contact( #Interlock_Entradas.AvisoPaleta_NXT_Manual_Av )
      Coil( #AvisoPaleta_NXT_Manual_AV )
   END_RUNG
   RUNG wire#w1
      Contact( #Interlock_Entradas.AvisoPaleta_NXT_Manual_Ret )
      Coil( #AvisoPaleta_NXT_Manual_Ret )
   END_RUNG
   RUNG wire#w1
      Contact( #PermisoPaleta_NXT_Manual_Av )
      Coil( #Interlock_Salidas.PermisoPaleta_NXT_Manual_Av )
   END_RUNG
   RUNG wire#w1
      Contact( #PermisoPaleta_NXT_Manual_Ret )
      Coil( #Interlock_Salidas.PermisoPaleta_NXT_Manual_Ret )
   END_RUNG
   // the same network as SCL:
   #AvisoPaleta_NXT_Manual_AV := "ON" AND #Interlock_Entradas.AvisoPaleta_NXT_Manual_Av;
   #AvisoPaleta_NXT_Manual_Ret := "ON" AND #Interlock_Entradas.AvisoPaleta_NXT_Manual_Ret;
   #Interlock_Salidas.PermisoPaleta_NXT_Manual_Av := "ON" AND #PermisoPaleta_NXT_Manual_Av;
   #Interlock_Salidas.PermisoPaleta_NXT_Manual_Ret := "ON" AND #PermisoPaleta_NXT_Manual_Ret;
END_REGION

NETWORK
TITLE = ----
//////////////////////////////////////////////////////////////////
/// Copia del Mckey de la Mesa de Salida de IKPAL

      CALL  UBLKMOV
      ( SRCBLK  := #Interlock_Entradas.MckeyPaletaSalida,
        RET_VAL := #ReturnValor,
        DSTBLK  := #Mckey_Paleta
      );

      L     #DBInstancia;
      T     #DBDestino;
      L     P##Mckey_Paleta;
      T     #P_Destino;
      SRD   3;
      L     #LongMckey;
      +I;
      L     1;
      -I;
      T     #OffsetDestino;

      L     #LongMckey;
Copia_MckeyPaleta:T     #Indice;

      OPN   DB [#DBDestino];
      L     DBB [#P_Destino];
      L     '0';
      +I;
      OPN   DB [#DBDestino];
      T     DBB [#P_Destino];

      L     #P_Destino;
      L     P#1.0;
      +D;
      T     #P_Destino;

      L     #Indice;
      LOOP  Copia_MckeyPaleta;

      CALL  "FC890_EtiqChar_EtiqDInt"
      ( DB_String   := #DBDestino,
        Long_String := #LongMckey,
        Offset_Ini  := #OffsetDestino,
        Valor       := #Valor
      );

      L     #Valor;
      T     #NumMckey_Paleta;


//////////////////////////////////////////////////////////////////
/// Copia de la Matricula de la Mesa de Salida de IKPAL

      CALL  UBLKMOV
      ( SRCBLK  := #Interlock_Entradas.MatriculaPaletaSalida,
        RET_VAL := #ReturnValor,
        DSTBLK  := #Matricula_Paleta
      );

      L     #DBInstancia;
      T     #DBOrigen;
      L     P##Matricula_Paleta;
      T     #P_Origen;

      L     #DBInstancia;
      T     #DBDestino;
      L     P##Matricula_Paleta;
      T     #P_Destino;

      L     #LongMatricula;
Copia_MatriculaPaleta:T     #Indice;

      OPN   DB [#DBOrigen];
      L     DBB [#P_Origen];
      L     '0';
      +I;
      OPN   DB [#DBDestino];
      T     DBB [#P_Destino];

      L     #P_Origen;
      L     P#1.0;
      +D;
      T     #P_Origen;

      L     #P_Destino;
      L     P#1.0;
      +D;
      T     #P_Destino;

      L     #Indice;
      LOOP  Copia_MatriculaPaleta;


//////////////////////////////////////////////////////////////////
/// Copia del Identificador de la UT de la Mesa de Salida de IKPAL

      L     #Interlock_Entradas.NumeroPaletaSalida;
      CAD;
      T     #IdentificadorUT_Paleta;



NETWORK
TITLE = Escritura de las Salidas
//////////////////////////////////////////////////////////////////////////////
/// Escritura de las Salidas

      SET;  // Comprobacion del Nodo
      AN    #Nodo_OK;
      JC    NoEscribirInterlock;

      CALL  UBLKMOV
      ( SRCBLK  := #P_L_Salidas,
        RET_VAL := #ReturnValor,
        DSTBLK  := #P_Salidas
      );


//////////////////////////////////////////////////////////////////////////////
/// Final Esctitura de las Salidas

NoEscribirInterlock:NOP   0;

      CALL  UBLKMOV
      ( SRCBLK  := #P_L_Salidas,
        RET_VAL := #ReturnValor,
        DSTBLK  := #P_DI_Salidas
      );  // Guardar el DB de Instancia




REGION Network 32: FINALIZAR - Guardar las Variables de Trabajo de la Mesa de Preformado
   RUNG wire#powerrail
      Move(in := #EstadoVIMesaPreformado, out1 => "DB900_Estado_Mesas".EstadoVI[#MesaPreformado])
   END_RUNG
   // the same network as SCL:
   "DB900_Estado_Mesas".EstadoVI[#MesaPreformado] := #EstadoVIMesaPreformado;
END_REGION

REGION Network 33: FINALIZAR - Guardar las Variables de Trabajo de la Mesa de Vacios
   RUNG wire#powerrail
      Move(in := #EstadoVIMesaVacios, out1 => "DB900_Estado_Mesas".EstadoVI[#MesaVacios])
   END_RUNG
   // the same network as SCL:
   "DB900_Estado_Mesas".EstadoVI[#MesaVacios] := #EstadoVIMesaVacios;
END_REGION

REGION Network 34: FINALIZAR - Guardar las Variables de Trabajo de la Mesa de Paleta
   RUNG wire#powerrail
      Move(in := #EstadoVIMesaPaleta, out1 => "DB900_Estado_Mesas".EstadoVI[#MesaPaleta])
   END_RUNG
   // the same network as SCL:
   "DB900_Estado_Mesas".EstadoVI[#MesaPaleta] := #EstadoVIMesaPaleta;
END_REGION
END_FUNCTION_BLOCK
